// TIA Portal V18 export
FUNCTION "AHUHeaterCtrl" : Void   // FC60303, LAD
{ S7_Optimized_Access := 'TRUE' }
VERSION : 0.1
// stored: AutoNumber false, IsIECCheckEnabled false, SetENOAutomatically false, UDAEnableTagReadback false
   VAR_INPUT
      UnitID : Int;
      DemandHeating : Real;
      FrostProtectionDemand : Real;
   END_VAR
   VAR_OUTPUT
      ValveAORequest : Real;
   END_VAR
BEGIN
END_FUNCTION
